// TIA Portal V19 export
TYPE "LEXCHANGETRAY_typePc_Monitor"
// stored: Access Published
   STRUCT
      status { S7_SetPoint := 'True'} : "LEXCHANGETRAY_typePc_Status";   // status
      cellsInfo { S7_SetPoint := 'True'} : "LEXCHANGETRAY_typeCellsMonitor";   // cellsinfo
      simulationed { S7_SetPoint := 'True'} : Bool;   // simulate
   END_STRUCT;
END_TYPE
